{attribute 'linkalways'} 
{attribute 'no_explicit_call' := 'This FB is a CLASS and must be accessed using methods or properties'}
{attribute 'enable_dynamic_creation'}
FUNCTION_BLOCK _WORD EXTENDS NumericDatatypeBase
VAR
	localData : WORD;
	activeData : REFERENCE TO WORD REF= localData;
END_VAR

PROPERTY PUBLIC Address : PVOID
GET
Address := ADR(activeData);
END_GET
END_PROPERTY

METHOD PUBLIC ClearReference
VAR_INPUT
END_VAR
activeData REF= localData;
END_METHOD

METHOD PUBLIC Clone : I_Datatype
VAR
    pClone : POINTER TO _WORD;
END_VAR
pClone := __NEW(_WORD(InitialValue := Value));
Clone := pClone^;
END_METHOD

METHOD FB_init : BOOL
VAR_INPUT
	bInitRetains : BOOL; // if TRUE, the retain variables are initialized (warm start / cold start)
	bInCopyCode : BOOL;  // if TRUE, the instance afterwards gets moved WORDo the copy code (online change)
	InitialValue : WORD;
END_VAR
localData := InitialValue;
END_METHOD

PROPERTY PUBLIC IsFloat : BOOL
GET
IsFloat := FALSE;
END_GET
END_PROPERTY

PROPERTY PUBLIC IsSigned : BOOL
GET
IsSigned := FALSE;
END_GET
END_PROPERTY

METHOD PUBLIC MakeReferenceTo
VAR_INPUT
	ReferenceTarget : REFERENCE TO WORD;
END_VAR
activeData REF= ReferenceTarget;
END_METHOD

PROPERTY PUBLIC MaxValue : WORD
GET
MaxValue :=  DatatypeLimits.WORD_MAX_VALUE;
END_GET
END_PROPERTY

PROPERTY PUBLIC MinValue : WORD
GET
MinValue := DatatypeLimits.WORD_MIN_VALUE;
END_GET
END_PROPERTY

METHOD PROTECTED SerializeMaxValue
VAR_INPUT
	Serializer : I_Serializer;
END_VAR
Serializer.AddWord(MaxValue);
END_METHOD

METHOD PROTECTED SerializeMinValue
VAR_INPUT
	Serializer : I_Serializer;
END_VAR
Serializer.AddWord(MinValue);
END_METHOD

METHOD PUBLIC SerializeWith
VAR_INPUT
	Serializer : I_Serializer;
END_VAR
Serializer.AddWord(activeData);
END_METHOD

PROPERTY PUBLIC Size : UDINT
GET
Size := SIZEOF(activeData);
END_GET
END_PROPERTY

METHOD TryDeserializeFrom : BOOL
VAR_INPUT
	Deserializer : I_Deserializer;
	Feedback : I_DeserializerFeedback;
END_VAR
TryDeserializeFrom := Deserializer.TryGetWord(activeData, Feedback);
END_METHOD

METHOD TryMakeReferenceTo : BOOL
VAR_INPUT
	Target : I_Datatype;
END_VAR
VAR
	pTargetData : POINTER TO WORD;
END_VAR
IF NOT (Target.TypeName = TypeName) THEN
	RETURN;
END_IF

pTargetData := Target.Address;
activeData REF= pTargetData^;
TryMakeReferenceTo := TRUE;
END_METHOD

PROPERTY PUBLIC TypeName : T_MAXSTRING
GET
TypeName := 'WORD';
END_GET
END_PROPERTY

PROPERTY PUBLIC Value : WORD
GET
Value := activeData;
END_GET
SET
activeData := Value;
END_SET
END_PROPERTY

END_FUNCTION_BLOCK

(* stored: Version 1.1.0.1, ProductVersion 3.1.4024.12
   POU _WORD: Id {d0df5d5f-5f73-44de-b259-1333c31f931d}, SpecialFunc None
   Folder Constructor: Id {834d5ad5-3f28-4dc0-8e98-0a08733c882d}
   Folder Protected: Id {0eb8423f-4e41-4145-8d48-cf18cfb15f8a}
   Property Address: Id {756d2378-fb99-457f-a9ff-9bda00e4192f}
   Get Get: Id {bd070509-c8ed-47d7-b7bf-ead1fac42360}
   Method ClearReference: Id {a8efd050-50b6-439b-97f5-5de554d92996}
   Method Clone: Id {925c1536-8da9-42d9-a001-a2effad3035c}
   Method FB_init: Id {8d4f9888-1fbd-47c7-bdc6-14c9ef7e73ce}
   Property IsFloat: Id {38b5d7ba-4eff-44c6-9c9f-7ab692c17933}
   Get Get: Id {db149071-8784-4256-b253-c419316678a8}
   Property IsSigned: Id {dd6fd2c2-fd73-416b-88a9-d1d06f96304e}
   Get Get: Id {e350b6a7-7f6d-4d84-849e-2ea436b4db50}
   Method MakeReferenceTo: Id {e40c9489-63c5-4da7-b7c6-14b92b878241}
   Property MaxValue: Id {779c2f15-cf65-4d03-8fef-92c3b5998ff1}
   Get Get: Id {80795371-e4f2-45a5-a02b-0760f092c2b3}
   Property MinValue: Id {9f5c1378-a49f-4661-97b2-360a09115292}
   Get Get: Id {d00f667d-253b-4bcb-ad65-40beaf23dd0b}
   Method SerializeMaxValue: Id {c47265b6-d098-4697-bdf8-6b219611c1a0}
   Method SerializeMinValue: Id {36eaa2aa-ebaf-4d5f-906f-d9f825eaa87d}
   Method SerializeWith: Id {5787a0f4-bdbb-4bfd-a299-7aa5b0f9b75f}
   Property Size: Id {8359033e-f446-4a6b-8300-5284ea1d2d31}
   Get Get: Id {11d88218-a391-4fc0-a436-bc22716332dd}
   Method TryDeserializeFrom: Id {a874291f-b4a2-45da-9197-930e58627d58}
   Method TryMakeReferenceTo: Id {00deb372-22af-4049-ad54-8cb491e6d3ad}
   Property TypeName: Id {42e30f31-1187-432c-a60f-3b1b2fcf5cc7}
   Get Get: Id {1113d29f-289d-493a-9efc-35a3c9852e26}
   Property Value: Id {4eafd79a-1247-497c-9696-ba0681ecad5b}
   Get Get: Id {eeebb207-39f4-4e06-a2c8-4aebb9d757dd}
   Set Set: Id {3dc23bcc-ce2d-489e-af29-247c99396ce0} *)
